PROGRAM MAIN
VAR
END_VAR

END_PROGRAM

(* stored: Version 1.1.0.1
   POU MAIN: Id {1668c7a5-c10d-4b27-a3e5-4fc8521ffe20} *)
